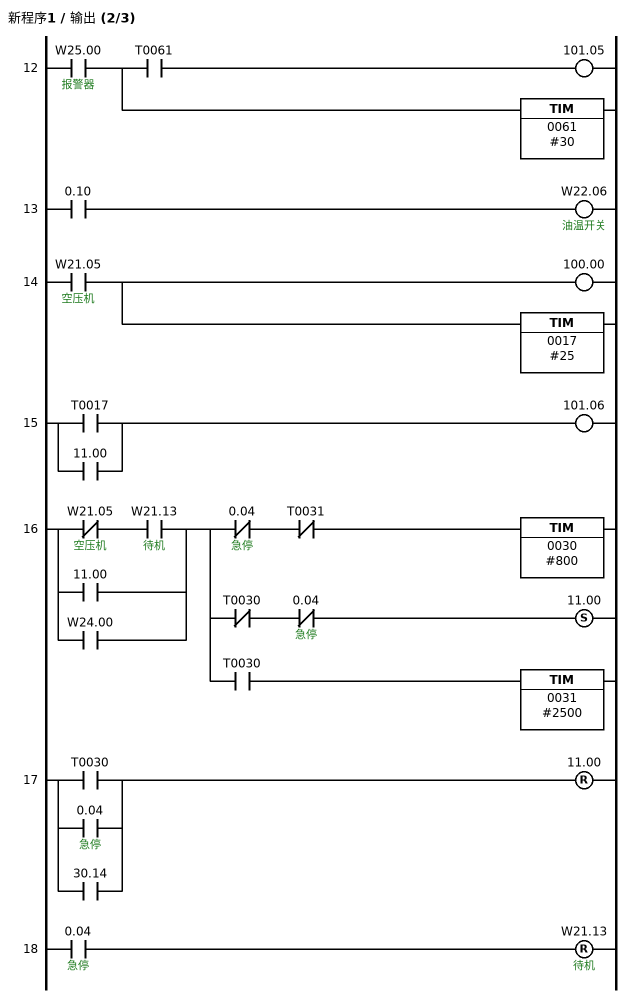
; [picture p24: 新程序1 / 输出, rungs 12-18]
; rung 12
LD W25.00  ; 报警器
OUT TR0
AND T0061
OUT 101.05
LD TR0
TIM 0061 #30
; rung 13
LD 0.10
OUT W22.06  ; 油温开关
; rung 14
LD W21.05  ; 空压机
OUT 100.00
TIM 0017 #25
; rung 15
LD T0017
OR 11.00
OUT 101.06
; rung 16
LDNOT W21.05  ; 空压机
AND W21.13  ; 待机
OR 11.00
OR W24.00
OUT TR0
ANDNOT 0.04  ; 急停
ANDNOT T0031
TIM 0030 #800
LD TR0
ANDNOT T0030
ANDNOT 0.04  ; 急停
SET 11.00
LD TR0
AND T0030
TIM 0031 #2500
; rung 17
LD T0030
OR 0.04  ; 急停
OR 30.14
RSET 11.00
; rung 18
LD 0.04  ; 急停
RSET W21.13  ; 待机

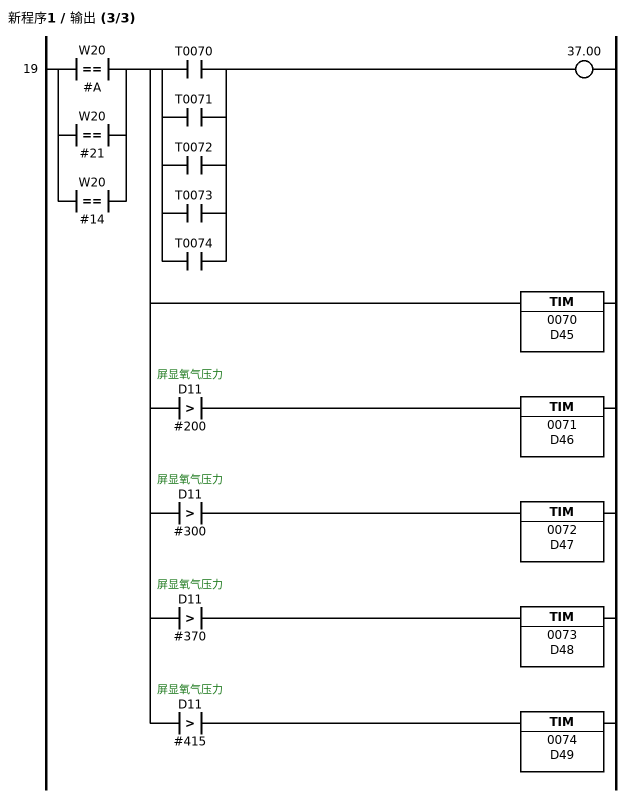
; rung 19
LD=(300) W20 #A
OR=(300) W20 #21
OR=(300) W20 #14
OUT TR0
LD T0070
OR T0071
OR T0072
OR T0073
OR T0074
ANDLD
OUT 37.00
LD TR0
TIM 0070 D45
AND>(320) D11 #200  ; 屏显氧气压力
TIM 0071 D46
LD TR0
AND>(320) D11 #300  ; 屏显氧气压力
TIM 0072 D47
LD TR0
AND>(320) D11 #370  ; 屏显氧气压力
TIM 0073 D48
LD TR0
AND>(320) D11 #415  ; 屏显氧气压力
TIM 0074 D49

### Section GPRS

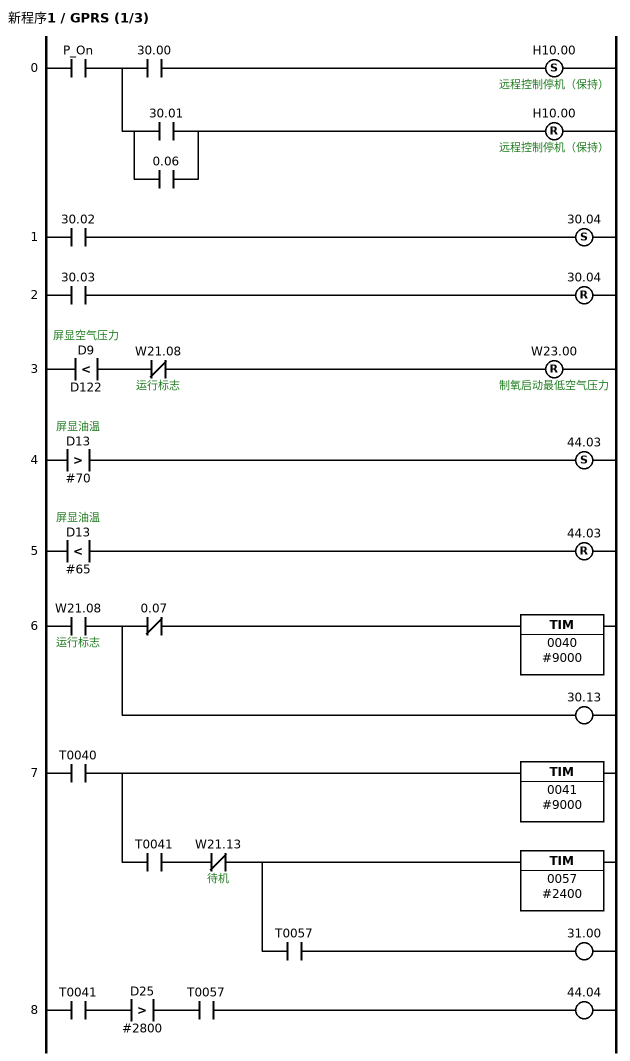
; rung 0
LD P_On
OUT TR0
AND 30.00
SET H10.00  ; 远程控制停机（保持）
LD TR0
LD 30.01
OR 0.06
ANDLD
RSET H10.00  ; 远程控制停机（保持）
; rung 1
LD 30.02
SET 30.04
; rung 2
LD 30.03
RSET 30.04
; rung 3
LD<(310) D9 D122  ; 屏显空气压力
ANDNOT W21.08  ; 运行标志
RSET W23.00  ; 制氧启动最低空气压力
; rung 4
LD>(320) D13 #70  ; 屏显油温
SET 44.03
; rung 5
LD<(310) D13 #65  ; 屏显油温
RSET 44.03
; rung 6
LD W21.08  ; 运行标志
OUT TR0
ANDNOT 0.07
TIM 0040 #9000
LD TR0
OUT 30.13
; rung 7
LD T0040
TIM 0041 #9000
AND T0041
ANDNOT W21.13  ; 待机
TIM 0057 #2400
AND T0057
OUT 31.00
; rung 8
LD T0041
AND>(320) D25 #2800
AND T0057
OUT 44.04

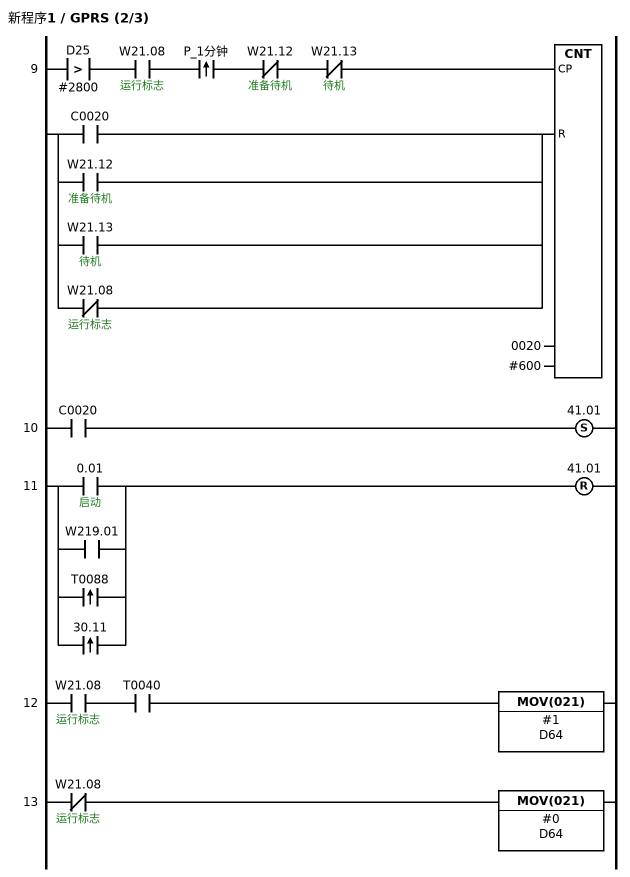
; rung 9
LD>(320) D25 #2800
AND W21.08  ; 运行标志
@AND P_1分钟
ANDNOT W21.12  ; 准备待机
ANDNOT W21.13  ; 待机
LD C0020
OR W21.12  ; 准备待机
OR W21.13  ; 待机
ORNOT W21.08  ; 运行标志
CNT 0020 #600
; rung 10
LD C0020
SET 41.01
; rung 11
LD 0.01  ; 启动
OR W219.01
@OR T0088
@OR 30.11
RSET 41.01
; rung 12
LD W21.08  ; 运行标志
AND T0040
MOV(021) #1 D64
; rung 13
LDNOT W21.08  ; 运行标志
MOV(021) #0 D64

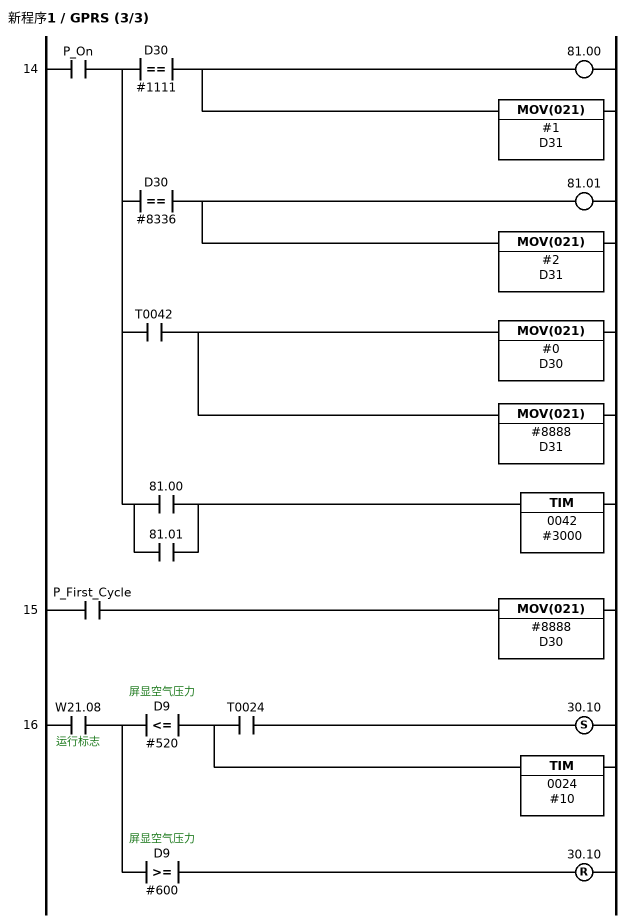
; rung 14
LD P_On
OUT TR0
AND=(300) D30 #1111
OUT 81.00
MOV(021) #1 D31
LD TR0
AND=(300) D30 #8336
OUT 81.01
MOV(021) #2 D31
LD TR0
AND T0042
MOV(021) #0 D30
MOV(021) #8888 D31
LD TR0
LD 81.00
OR 81.01
ANDLD
TIM 0042 #3000
; rung 15
LD P_First_Cycle
MOV(021) #8888 D30
; rung 16
LD W21.08  ; 运行标志
OUT TR0
AND<=(315) D9 #520  ; 屏显空气压力
OUT TR1
AND T0024
SET 30.10
LD TR1
TIM 0024 #10
LD TR0
AND>=(325) D9 #600  ; 屏显空气压力
RSET 30.10

### Section 结束
; rung 0
END(001)